// Implicitly generated code : DO NOT EDIT
FUNCTION CheckBounds : DINT
VAR_INPUT
    index, lower, upper: DINT;
END_VAR

// Implicitly generated code : Only an Implementation suggestion
{noflow}
IF  index < lower THEN
    CheckBounds := lower;
ELSIF  index > upper THEN
    CheckBounds := upper;
ELSE
    CheckBounds := index;
END_IF
{flow}

END_FUNCTION

(* stored: Version 1.1.0.1
   POU CheckBounds: Id {a57f8efa-1f2c-4ddd-893c-0e58639bc631}, SpecialFunc CheckBounds *)
